{attribute addProperty BoxType "EL3403-0000-0018"}
{attribute addProperty Id "PM_Inputs_ChannelAT %I*ARRAY[0..2] OF PM_Inputs_Channel_2B79FE26456570PM_Status_dataAT %I*PM_Status_data_CC42570F4050PM_Outputs_ChannelAT %Q*ARRAY[0..2] OF PM_Outputs_Channel_A1108FBB2430WcStateAT %I*WcState_F855686C1620InfoDataAT %I*InfoData_BC63D37F80100"}
{attribute addProperty CRC "3182249553"}
{attribute addProperty SizeInBites "616"}
{attribute addProperty SizeInBytes "77"}
TYPE EL3403_0856E9FD :
STRUCT
	{attribute addProperty Name "PM_Inputs_Channel"}
	PM_Inputs_Channel : ARRAY[0..2] OF PM_Inputs_Channel_2B79FE26;
	{attribute addProperty Name "PM_Status_data"}
	PM_Status_data : PM_Status_data_CC42570F;
	{attribute addProperty Name "PM_Outputs_Channel"}
	PM_Outputs_Channel : ARRAY[0..2] OF PM_Outputs_Channel_A1108FBB;
	{attribute addProperty Name "WcState"}
	WcState : WcState_F855686C;
	{attribute addProperty Name "InfoData"}
	InfoData : InfoData_BC63D37F;
END_STRUCT
END_TYPE

(* stored: Version 1.2.0.0, ProductVersion 3.1.4024.9
   DUT EL3403_0856E9FD: Id {690dc85e-54eb-4ff4-a4f6-7ca3737a4b91} *)
